# EPICS autosave request: support/dxp/2-9/dxpApp/Db/dxpMED_settings.req
$(P)PresetReal
$(P)PresetLive
$(P)StatusAll.SCAN
$(P)ReadAll.SCAN
$(P)ReadDXPs.SCAN
$(P)ReadDXPBaselines.SCAN
$(P)BaselineHistoryTimes
$(P)TraceWaits
$(P)EnableClientWait
